SUBAPPLICATION Uebung_007d4 (* Blinker mit E_CYCLE und E_T_FF *)
  (* Standard: 61499-2; Description: Copyright (c) 2023 Meisterschulen am Ostbahnhof This program and the accompanying materials are made available under the terms of the Eclipse Public License 2.0 which is available at https://www.eclipse.org/legal/epl-2.0/ SPDX-License-Identifier: EPL-2.0 *)
  (* Version 1.0, 2023-10-23, Franz Höpfinger, Meisterschulen am Ostbahnhof, initial API and implementation and/or initial documentation *)
  PACKAGE Uebungen;
  IMPORT logiBUS::io::DQ::logiBUS_DO::Output_Q1;
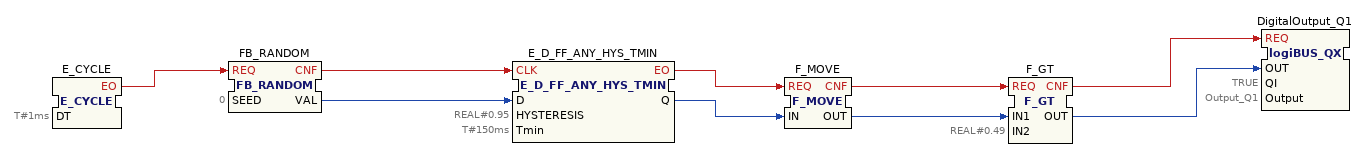
  FBS
    DigitalOutput_Q1 : logiBUS::io::DQ::logiBUS_QX(QI := TRUE, Output := Output_Q1);
    E_CYCLE : iec61499::events::E_CYCLE(DT := T#1ms);
    FB_RANDOM : eclipse4diac::utils::FB_RANDOM(SEED := 0);
    F_GT : iec61131::comparison::F_GT(IN2 := REAL#0.49);
    E_D_FF_ANY_HYS_TMIN : logiBUS::signalprocessing::hysteresis::E_D_FF_ANY_HYS_TMIN(HYSTERESIS := REAL#0.95, Tmin := T#150ms);
    F_MOVE : iec61131::selection::F_MOVE; {SET_ATTRIBUTE(DataType, REAL)}
  END_FBS
  EVENT_CONNECTIONS
    E_CYCLE.EO TO FB_RANDOM.REQ;
    FB_RANDOM.CNF TO E_D_FF_ANY_HYS_TMIN.CLK;
    F_GT.CNF TO DigitalOutput_Q1.REQ;
    E_D_FF_ANY_HYS_TMIN.EO TO F_MOVE.REQ;
    F_MOVE.CNF TO F_GT.REQ;
  END_CONNECTIONS
  DATA_CONNECTIONS
    FB_RANDOM.VAL TO E_D_FF_ANY_HYS_TMIN.D;
    F_GT.OUT TO DigitalOutput_Q1.OUT;
    E_D_FF_ANY_HYS_TMIN.Q TO F_MOVE.IN;
    F_MOVE.OUT TO F_GT.IN1;
  END_CONNECTIONS
END_SUBAPPLICATION
